{region '#Template'}
	{attribute 'Version' := '1.0.0.0'}
	{attribute 'Tags' := '"LCID": "1031", "Text": "DUT, Plant, AC, Setpoint"'}
	{attribute 'Tags' := '"LCID": "1033", "Text": "DUT, Plant, AC, Setpoint"'}
	{attribute 'Description' := '"LCID": "1031", "Text": "Auswahl Sollwert Energie Rückgewinnung"'}
	{attribute 'Description' := '"LCID": "1033", "Text": "Selection setpoint energy recovery"'}
{endregion}

{attribute 'qualified_only'}
TYPE E_BA_AC_SelSpErc :
(
	eAction				:= 1,	//	E_BA_Action.eDirect = SpCol, E_BA_Action.eReverse = SpHtg, 
	eAverageHtgCol		:= 2	
) UDINT;
END_TYPE

(* stored: Version 1.1.0.1, ProductVersion 3.1.4024.9
   DUT E_BA_AC_SelSpErc: Id {b88c1475-160e-4cca-b1fd-86a3d96b1ebb} *)
